(* IEC 61131-3 sources: Industry-PLC-LLM/data/PLCBEAD_repo/PLCBEAD_PLCEmbed-main/PLC-BEAD/Source/GEB/Network__BUFFER_UPPERCASE_NW, 1 file *)

(* ---- _BUFFER_UPPERCASE_NW.ST ---- *)
TYPE
  oscat_NW_BUF_LONG  : ARRAY [0..4095] OF BYTE;
END_TYPE

FUNCTION SETUP_EXTENDED_ASCII:BOOL
	VAR_INPUT
		X :	BOOL;
	END_VAR

	SETUP_EXTENDED_ASCII := X OR TRUE;
END_FUNCTION

FUNCTION TO_UPPER:BYTE

	VAR_INPUT
		IN :	BYTE;
	END_VAR

	IF IN > BYTE#96 AND IN < BYTE#123 THEN
	TO_UPPER := IN AND BYTE#16#DF;
	ELSIF IN > BYTE#223 AND IN <> BYTE#247 AND IN <> BYTE#255 AND SETUP_EXTENDED_ASCII(FALSE) THEN
	TO_UPPER := IN AND BYTE#16#DF;
	ELSE
	TO_UPPER := IN;
	END_IF;

END_FUNCTION

FUNCTION_BLOCK _BUFFER_UPPERCASE_NW
	VAR_INPUT
		SIZE :	UINT;
	END_VAR

	VAR_OUTPUT
		_BUFFER_UPPERCASE :	BOOL;
	END_VAR

	VAR_IN_OUT
		PT :	oscat_NW_BUF_LONG;
	END_VAR

	VAR
		POS :	INT;
		SIZE2 :	INT;
	END_VAR

	POS := 0;
	SIZE2 := UINT_TO_INT(SIZE);

	WHILE POS < SIZE2 DO
		PT[POS] := TO_UPPER(PT[POS]);
		POS := POS + 1;
	END_WHILE;

	_BUFFER_UPPERCASE := TRUE;

END_FUNCTION_BLOCK

PROGRAM program0
  VAR
	SIZE :	UINT;

	_BUFFER_UPPERCASE :	BOOL;

	PT :	oscat_NW_BUF_LONG;

	func_block : _BUFFER_UPPERCASE_NW;
  END_VAR
	func_block.SIZE  :=SIZE ;
	func_block.PT  :=PT ;
	func_block();
	PT := func_block.PT;
	_BUFFER_UPPERCASE := func_block._BUFFER_UPPERCASE;
END_PROGRAM
